FUNCTION_BLOCK E_DEFAULT_PERMIT (* permissive propagation of an event *)
  (* Standard: 61499-1 Annex A; Description: Copyright (c) 2017 fortiss GmbH This program and the accompanying materials are made available under the terms of the Eclipse Public License 2.0 which is available at https://www.eclipse.org/legal/epl-2.0/ SPDX-License-Identifier: EPL-2.0 *)
  (* Version 1.0, 2017-09-20, Alois Zoitl, fortiss GmbH, initial API and implementation and/or initial documentation *)
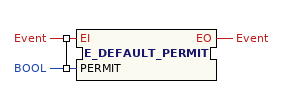
  EVENT_INPUT
    EI WITH PERMIT;
  END_EVENT
  EVENT_OUTPUT
    EO;
  END_EVENT
  VAR_INPUT
    PERMIT : BOOL := TRUE;
  END_VAR
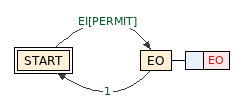
  EC_STATES
    START; (* Initial State *)
    EO : -> EO; (* Event propagration permited *)
  END_STATES
  EC_TRANSITIONS
    START TO EO := EI[PERMIT];
    EO TO START := 1;
  END_TRANSITIONS
END_FUNCTION_BLOCK
